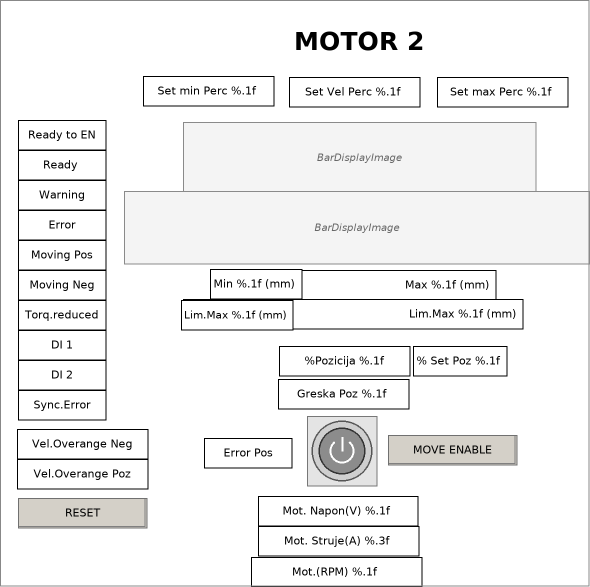
VISUALIZATION Visualization2  // 590x587
    Rectangle (210,270 286x30), "Max %.1f (mm)", text variable: MAIN.FB_DC_MOTOR2.rRadno_Max_Pos
        OnMouseDown: write the text variable via Default, min 0, max 100
    PowerSwitch (307,416 70x70), variable: MAIN.bMotorOn_M2, behaviour: TOGGLE, style: Switch-PowerSwitch-Gray
    Rectangle (143,76 131x30), "Set min Perc %.1f", text variable: MAIN.rSetpointTarget_MinM2
        OnMouseDown: write the text variable via Default, min 0, max 100
    Rectangle (437,77 131x30), "Set max Perc %.1f", text variable: MAIN.rSetpointTarget_MaxM2
        OnMouseDown: write the text variable via Default, min 0, max 100
    Rectangle (279,346 131x30), "%Pozicija %.1f", text variable: MAIN.rPotFeedback_Radno_PercM2
    Rectangle (289,77 131x30), "Set Vel Perc %.1f", text variable: MAIN.rMaxVelocityM2
        OnMouseDown: write the text variable via Default, min 0, max 120
    Rectangle (278,379 131x30), "Greska Poz %.1f", text variable: MAIN.rErrorM2, colour toggle: MAIN.bInDeadband_M2
    Rectangle (258,496 160x30), "Mot. Napon(V) %.1f", text variable: MAIN.rMotorVoltageM2
    Rectangle (258,526 161x30), "Mot. Struje(A) %.3f", text variable: MAIN.rMotorCurrentM2
    Rectangle (413,346 94x30), "% Set Poz %.1f", text variable: MAIN.rSetpointTarget_M2
    Rectangle (251,557 171x30), "Mot.(RPM) %.1f", text variable: MAIN.rActualVelocityRPM_M2
    Rectangle (17,429 131x30), "Vel.Overange Neg", colour toggle: MAIN.FB_DC_MOTOR2.bSetVelOverNeg
    Rectangle (17,459 131x30), "Vel.Overange Poz", colour toggle: MAIN.FB_DC_MOTOR2.bSetVelOverPoz
    Button (18,498 129x30), "RESET"
        tap MAIN.bHMI_RESET_M2
    Rectangle (18,120 88x30), "Ready to EN", colour toggle: bReadyToEnable_M2
    Rectangle (18,150 88x30), "Ready", colour toggle: bReady_M2
    Rectangle (18,180 88x30), "Warning", colour toggle: bWarning_M2
    Rectangle (18,210 88x30), "Error", colour toggle: bError_M2
    Rectangle (18,240 88x30), "Moving Pos", colour toggle: bMovingPositive_M2
    Rectangle (18,270 88x30), "Moving Neg", colour toggle: bMovingNegative_M2
    Rectangle (18,300 88x30), "Torq.reduced", colour toggle: bTorqueReduced_M2
    Rectangle (18,330 88x30), "DI 1", colour toggle: bDigitalInput1_M2
    Rectangle (18,360 88x30), "DI 2", colour toggle: bDigitalInput2_M2
    Rectangle (18,390 88x30), "Sync.Error", colour toggle: bSyncError_M2
    Button (388,435 129x30), "MOVE ENABLE", colour toggle: MAIN.bMove_M2
        toggle MAIN.bMove_M2
    BarDisplayImage (183,122 353x71), value: MAIN.rPotFeedback_Radno_PercM2, style: BarDisplayImage-Gray, scale format: %.1f, scale 0..100
        p518627256: %
    BarDisplayImage (124,191 466x73), value: MAIN.FB_DC_MOTOR2.rLinearPosition, style: BarDisplayImage-Gray, scale format: %.1f, scale 0..80
        p518627256: mm
    Rectangle (210,269 92x30), "Min %.1f (mm)", text variable: MAIN.FB_DC_MOTOR2.rRadno_Min_Pos
        OnMouseDown: write the text variable via Default, min 0, max 100
    Rectangle (183,299 340x30), "Lim.Max %.1f (mm)", text variable: MAIN.FB_DC_MOTOR2.rLinearPosition_LimMAx, colour toggle: MAIN.bErrorLimitPosMax_M2
        OnMouseDown: write the text variable via Default, min 0, max 100
    Rectangle (181,300 112x30), "Lim.Max %.1f (mm)", text variable: MAIN.FB_DC_MOTOR2.rLinearPosition_LimMin, colour toggle: MAIN.bErrorLimitPosMin_M2
        OnMouseDown: write the text variable via Default, min 0, max 100
    Label (148,26 423x30), "MOTOR 2"
    Rectangle (204,438 88x30), "Error Pos", colour toggle: MAIN.bERROR_POS_M2
END_VISUALIZATION

(* stored: Version 1.1.0.1, ProductVersion 3.1.4024.15
   Visu Visualization2: Id {a7557ec1-9a19-4383-8ebd-912f44bb219e} *)
